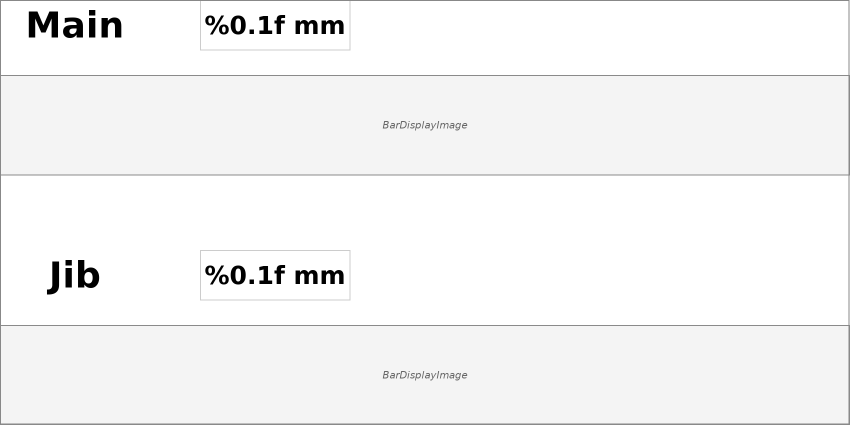
VISUALIZATION VISU_Position  // 850x425
    BarDisplayImage (0,75 850x100), value: fMain_Position_mm, style: BarDisplayImage-Gray, scale format: %.1f, scale 0..800
    Textfield (0,0 150x50), "Main"
    Textfield (0,250 150x50), "Jib"
    BarDisplayImage (0,325 850x100), value: fJib_Position_mm, style: BarDisplayImage-Gray, scale format: %.1f, scale 0..900
    Textfield (200,0 150x50), "%0.1f mm", text variable: fMain_Position_mm
    Textfield (200,250 150x50), "%0.1f mm", text variable: fJib_Position_mm
END_VISUALIZATION

(* stored: Version 1.1.0.1
   Visu VISU_Position: Id {79ff9d63-17a5-42f5-9820-d1a986dfeac7} *)
